(* IEC 61131-3 sources: Industry-PLC-LLM/data/PLCBEAD_repo/PLCBEAD_PLCEmbed-main/PLC-BEAD/Source/GEB/FRMP_B, 1 file *)

(* ---- FRMP_B.ST ---- *)
FUNCTION FRMP_B:BYTE

	VAR_INPUT
		START :	BYTE;
		DIR :	BOOL;
		TD :	TIME;
		TR :	TIME;
	END_VAR

	IF TD < TR THEN
		FRMP_B := MIN(UDINT_TO_BYTE(DWORD_TO_UDINT(SHL(TIME_TO_DWORD(TD), 8)) / TIME_TO_UDINT(TR)), SEL(DIR, START, USINT_TO_BYTE(USINT#255 - BYTE_TO_USINT(START))));
		IF DIR THEN
			FRMP_B := USINT_TO_BYTE(BYTE_TO_USINT(START) + BYTE_TO_USINT(FRMP_B));
		ELSE
			FRMP_B := USINT_TO_BYTE(BYTE_TO_USINT(START) - BYTE_TO_USINT(FRMP_B));
		END_IF;
	ELSE
		FRMP_B := SEL(DIR, BYTE#0, BYTE#255);
	END_IF;
END_FUNCTION

PROGRAM program0
  VAR
    LocalVar0 : BYTE;
	LocalVaR1  : BOOL;
	LocalVaR2 : TIME;
	LocalVar3 : TIME;
    LocalOUT  : BYTE;
  END_VAR

  LocalOUT := FRMP_B(LocalVar0, LocalVaR1 , LocalVaR2,LocalVar3);
END_PROGRAM
